// TIA Portal V15.1 export
// export: Created 2019-08-14T06:26:11.8498234Z, ExportSetting None, DisplayName Totally Integrated Automation Portal, DisplayVersion V15.1, DisplayName TIA Portal Openness, DisplayVersion V15.1, DisplayName STEP 7 Professional, DisplayVersion V15.1, DisplayName STEP 7 Safety, DisplayVersion V15.1, DisplayName WinCC Advanced, DisplayVersion V15.1
FUNCTION_BLOCK "#SKILL_NAME#_Start"   // FB14, SCL
{ S7_Optimized_Access := 'TRUE' }
// stored: MemoryReserve 100, SetENOAutomatically False
   VAR_INPUT
      ModulToSkill { ExternalAccessible := 'False'; ExternalVisible := 'False'; ExternalWritable := 'False'} : "typeModulSkillInterface_IN";
      SkillToModul { ExternalAccessible := 'False'; ExternalVisible := 'False'; ExternalWritable := 'False'} : "typeModulSkillInterface_OUT";
   END_VAR
   VAR_IN_OUT
      StartSkill : Bool;
      Parameter : "type#SKILL_NAME#StartParameter_In";
   END_VAR
   VAR
      OPC_UA_ServerMethodPre_Instance : OPC_UA_ServerMethodPre;
      OPC_UA_ServerMethodPost_Instance : OPC_UA_ServerMethodPost;
      UAMethod_InParameters : "type#SKILL_NAME#StartParameter_In";
      UAMethod_OutParameters : "type#SKILL_NAME#StartParameter_Out";
      UAMethod : "UA_Method_Handle";
   END_VAR
   VAR_TEMP
      Temp : Bool;
   END_VAR
BEGIN
   REGION PRE
       IF #UAMethod.Started = FALSE AND #UAMethod.Finished = FALSE THEN

           #OPC_UA_ServerMethodPre_Instance(Busy => #UAMethod.Pre.Busy,
                                            Done => #UAMethod.Pre.Done,
                                            Status => #UAMethod.Pre.Status,
                                            Error => #UAMethod.Pre.Error,
                                            UAMethod_Called => #UAMethod.Called,
                                            UAMethod_InParameters := #UAMethod_InParameters);

           IF #UAMethod.Pre.Error THEN
               #UAMethod.ErrorMessage := WString#'Error at OPC_UA_ServerMethodPre';
           END_IF;

           IF #UAMethod.Pre.Done AND #UAMethod.Called THEN
               #UAMethod.Started := TRUE;
               #UAMethod.ErrorMessage := WString#'';
           END_IF;

       END_IF;
   END_REGION

   REGION FUNCTIONALITY 

       IF #UAMethod.Started THEN
           (*
           // Enter User Code here
           //  - Check state of modul and skill control
           //  - Check incomming parameters
           // 
           *)


           // submit parameter and start to main skill FB
           // parameter is skill dependent
           #Parameter := #UAMethod_InParameters;
           #StartSkill := TRUE;

           #UAMethod.Result := 16#0;
           #UAMethod.ErrorMessage := WString#'';

           #UAMethod.Finished := TRUE;
           #UAMethod.Started := FALSE;
       END_IF;

   END_REGION


   REGION POST
       IF #UAMethod.Finished = TRUE THEN

           #OPC_UA_ServerMethodPost_Instance(UAMethod_Result := #UAMethod.Result,
                                             UAMethod_Finished := #UAMethod.Finished,
                                             Busy => #UAMethod.Post.Busy,
                                             Done => #UAMethod.Post.Done,
                                             Error => #UAMethod.Post.Error,
                                             Status => #UAMethod.Post.Status,
                                             UAMethod_OutParameters := #UAMethod_OutParameters);

           IF #UAMethod.Post.Error = TRUE THEN
               #StartSkill := FALSE;

               #UAMethod.ErrorMessage := WString#'Error at OPC_UA_ServerMethodPost';
               #UAMethod.Finished := FALSE;
           END_IF;

           IF #UAMethod.Post.Done = TRUE THEN
               #StartSkill := FALSE;
               #UAMethod.Finished := FALSE;
           END_IF;

       END_IF;

   END_REGION
END_FUNCTION_BLOCK
